% RSLogix 500 project FILLING STATION.RSS, saved by version 8.30.00.16 %
PROJECT "SIM_PLC"    % processor: Bul.1763 MicroLogix 1100 Series B %

PROGRAM FILES
  LAD 2 "MAIN"  4 rungs
  LAD 3 "INPUTS"  5 rungs
  LAD 4 "OUTPUTS"  4 rungs
  LAD 5 "CTRL LOGIC"  13 rungs

DATA FILES
  O0 OUTPUT  5 elements
  I1 INPUT  7 elements
  S2 STATUS  66 elements
  B3 BINARY  1 elements
  T4 TIMER  1 elements
  C5 COUNTER  1 elements
  R6 CONTROL  1 elements
  N7 INTEGER  1 elements
  F8 FLOAT  1 elements

LADDER 2 "MAIN"
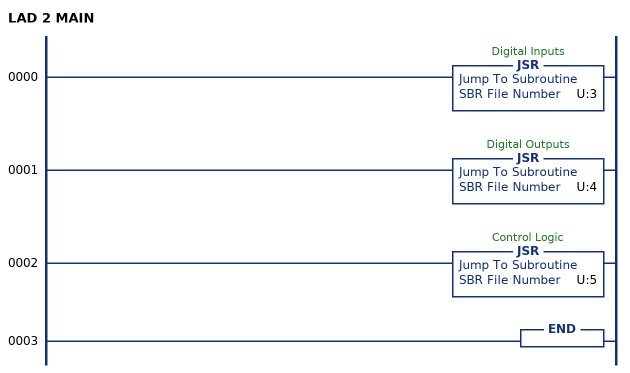
% Rung: 0 %
SOR JSR U:3 EOR
%   U:3  "Digital Inputs" %
% Rung: 1 %
SOR JSR U:4 EOR
%   U:4  "Digital Outputs" %
% Rung: 2 %
SOR JSR U:5 EOR
%   U:5  "Control Logic" %
% Rung: 3 %
SOR END EOR

LADDER 3 "INPUTS"
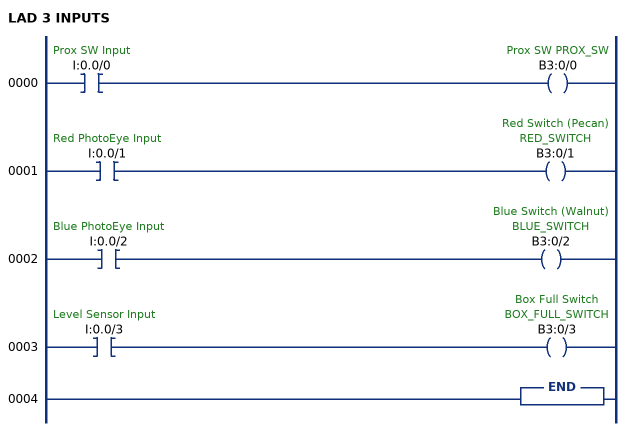
% Rung: 0 %
SOR XIC I:0.0/0 OTE B3:0/0 EOR
%   I:0.0/0  "Prox SW Input" %
%   B3:0/0  PROX_SW  "Prox SW" %
% Rung: 1 %
SOR XIC I:0.0/1 OTE B3:0/1 EOR
%   I:0.0/1  "Red PhotoEye Input" %
%   B3:0/1  RED_SWITCH  "Red Switch (Pecan)" %
% Rung: 2 %
SOR XIC I:0.0/2 OTE B3:0/2 EOR
%   I:0.0/2  "Blue PhotoEye Input" %
%   B3:0/2  BLUE_SWITCH  "Blue Switch (Walnut)" %
% Rung: 3 %
SOR XIC I:0.0/3 OTE B3:0/3 EOR
%   I:0.0/3  "Level Sensor Input" %
%   B3:0/3  BOX_FULL_SWITCH  "Box Full Switch" %
% Rung: 4 %
SOR END EOR

LADDER 4 "OUTPUTS"
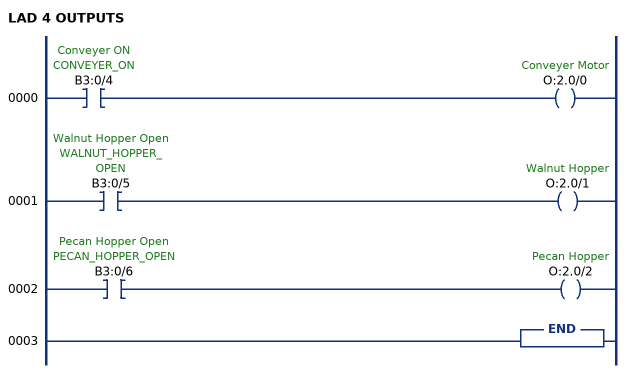
% Rung: 0 %
SOR XIC B3:0/4 OTE O:2.0/0 EOR
%   B3:0/4  CONVEYER_ON  "Conveyer ON" %
%   O:2.0/0  "Conveyer Motor" %
% Rung: 1 %
SOR XIC B3:0/5 OTE O:2.0/1 EOR
%   B3:0/5  WALNUT_HOPPER_OPEN  "Walnut Hopper Open" %
%   O:2.0/1  "Walnut Hopper" %
% Rung: 2 %
SOR XIC B3:0/6 OTE O:2.0/2 EOR
%   B3:0/6  PECAN_HOPPER_OPEN  "Pecan Hopper Open" %
%   O:2.0/2  "Pecan Hopper" %
% Rung: 3 %
SOR END EOR

LADDER 5 "CTRL LOGIC"
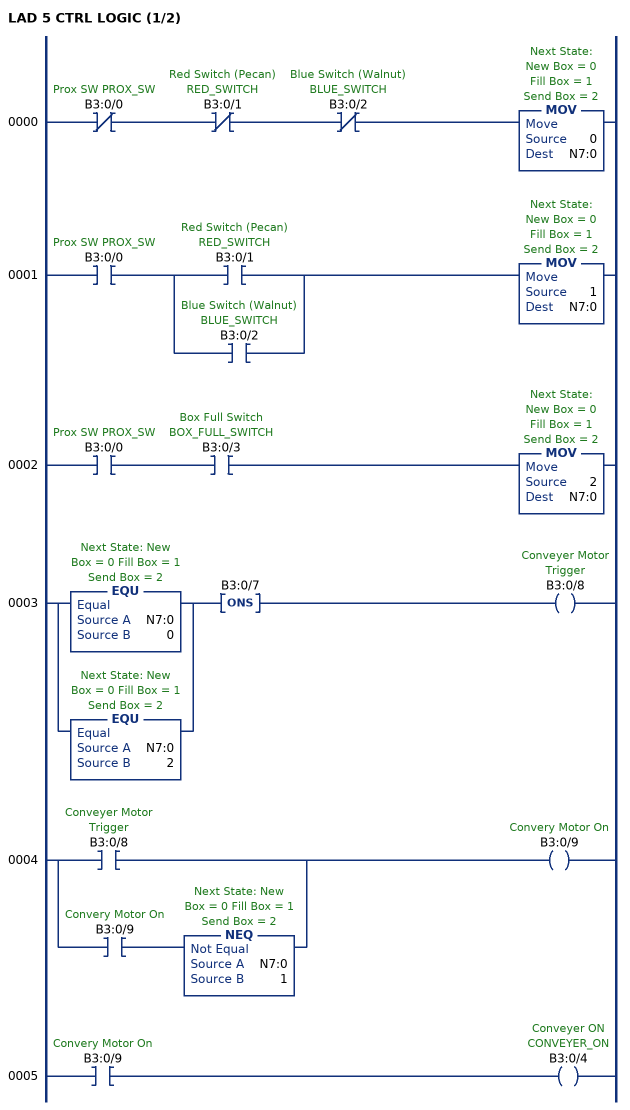
% Rung: 0 %
SOR XIO B3:0/0 XIO B3:0/1 XIO B3:0/2 MOV 0 N7:0 EOR
%   B3:0/0  PROX_SW  "Prox SW" %
%   B3:0/1  RED_SWITCH  "Red Switch (Pecan)" %
%   B3:0/2  BLUE_SWITCH  "Blue Switch (Walnut)" %
%   N7:0  "Next State: New Box = 0 Fill Box = 1 Send Box = 2" %
% Rung: 1 %
SOR XIC B3:0/0 BST XIC B3:0/1 NXB XIC B3:0/2 BND MOV 1 N7:0 EOR
%   B3:0/0  PROX_SW  "Prox SW" %
%   B3:0/1  RED_SWITCH  "Red Switch (Pecan)" %
%   B3:0/2  BLUE_SWITCH  "Blue Switch (Walnut)" %
%   N7:0  "Next State: New Box = 0 Fill Box = 1 Send Box = 2" %
% Rung: 2 %
SOR XIC B3:0/0 XIC B3:0/3 MOV 2 N7:0 EOR
%   B3:0/0  PROX_SW  "Prox SW" %
%   B3:0/3  BOX_FULL_SWITCH  "Box Full Switch" %
%   N7:0  "Next State: New Box = 0 Fill Box = 1 Send Box = 2" %
% Rung: 3 %
SOR BST EQU N7:0 0 NXB EQU N7:0 2 BND ONS B3:0/7 OTE B3:0/8 EOR
%   N7:0  "Next State: New Box = 0 Fill Box = 1 Send Box = 2" %
%   B3:0/8  "Conveyer Motor Trigger" %
% Rung: 4 %
SOR BST XIC B3:0/8 NXB XIC B3:0/9 NEQ N7:0 1 BND OTE B3:0/9 EOR
%   B3:0/8  "Conveyer Motor Trigger" %
%   B3:0/9  "Convery Motor On" %
%   N7:0  "Next State: New Box = 0 Fill Box = 1 Send Box = 2" %
% Rung: 5 %
SOR XIC B3:0/9 OTE B3:0/4 EOR
%   B3:0/9  "Convery Motor On" %
%   B3:0/4  CONVEYER_ON  "Conveyer ON" %

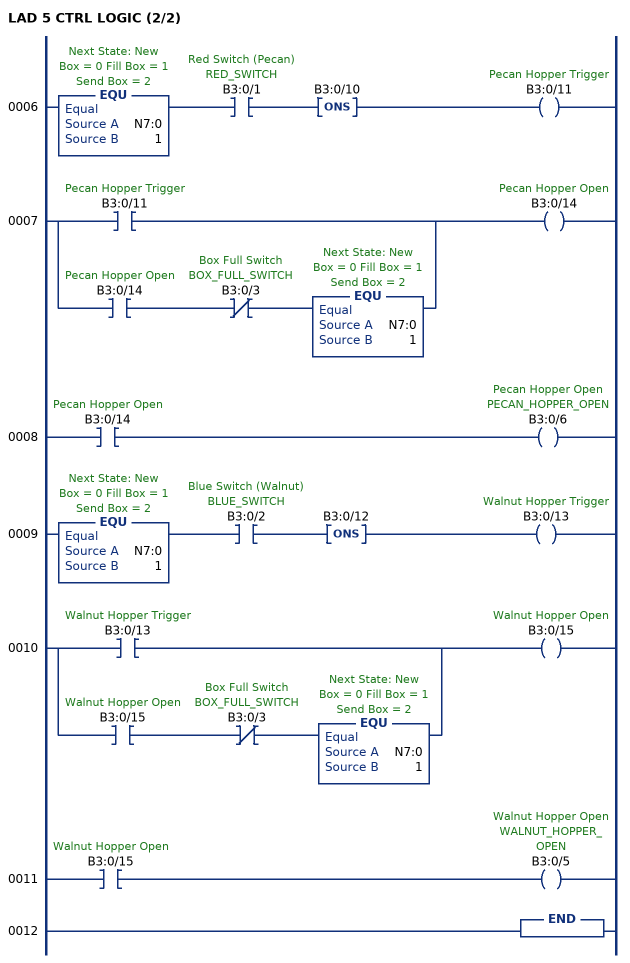
% Rung: 6 %
SOR EQU N7:0 1 XIC B3:0/1 ONS B3:0/10 OTE B3:0/11 EOR
%   N7:0  "Next State: New Box = 0 Fill Box = 1 Send Box = 2" %
%   B3:0/1  RED_SWITCH  "Red Switch (Pecan)" %
%   B3:0/11  "Pecan Hopper Trigger" %
% Rung: 7 %
SOR BST XIC B3:0/11 NXB XIC B3:0/14 XIO B3:0/3 EQU N7:0 1 BND OTE B3:0/14 EOR
%   B3:0/11  "Pecan Hopper Trigger" %
%   B3:0/14  "Pecan Hopper Open" %
%   B3:0/3  BOX_FULL_SWITCH  "Box Full Switch" %
%   N7:0  "Next State: New Box = 0 Fill Box = 1 Send Box = 2" %
% Rung: 8 %
SOR XIC B3:0/14 OTE B3:0/6 EOR
%   B3:0/14  "Pecan Hopper Open" %
%   B3:0/6  PECAN_HOPPER_OPEN  "Pecan Hopper Open" %
% Rung: 9 %
SOR EQU N7:0 1 XIC B3:0/2 ONS B3:0/12 OTE B3:0/13 EOR
%   N7:0  "Next State: New Box = 0 Fill Box = 1 Send Box = 2" %
%   B3:0/2  BLUE_SWITCH  "Blue Switch (Walnut)" %
%   B3:0/13  "Walnut Hopper Trigger" %
% Rung: 10 %
SOR BST XIC B3:0/13 NXB XIC B3:0/15 XIO B3:0/3 EQU N7:0 1 BND OTE B3:0/15 EOR
%   B3:0/13  "Walnut Hopper Trigger" %
%   B3:0/15  "Walnut Hopper Open" %
%   B3:0/3  BOX_FULL_SWITCH  "Box Full Switch" %
%   N7:0  "Next State: New Box = 0 Fill Box = 1 Send Box = 2" %
% Rung: 11 %
SOR XIC B3:0/15 OTE B3:0/5 EOR
%   B3:0/15  "Walnut Hopper Open" %
%   B3:0/5  WALNUT_HOPPER_OPEN  "Walnut Hopper Open" %
% Rung: 12 %
SOR END EOR

OTHER DOCUMENTED ADDRESSES
  PFILE:3  "Inputs"
  T4:0/DN  "Prox SW Closed"
  T4:1/DN  "Pecan Box Present"
  T4:2/DN  "Walnut Hopper Open"

DATA TABLE (non-zero values as saved)
DATA B3
% B3:0 % 0X0009
DATA T4
% .PRE .ACC %
% T4:0 % 5 5
